{attribute 'GeneratedUsingTerminal: EL3024-0000-0019'}
{attribute addProperty BoxType "EL3024-0000-0019"}
{attribute addProperty Id "StatusAT %I*Status_F2CE6D917ValueAT %I*INT2"}
{attribute addProperty CRC "1245267073"}
{attribute addProperty Size "9"}
TYPE AI_Standard_Channel_4A394481 EXTENDS InputBase_8311D824 :
STRUCT
	{attribute addProperty Name "Status"}
	Status AT %I* : Status_F2CE6D91;
	{attribute addProperty Name "Value"}
	Value AT %I* : INT;
END_STRUCT
END_TYPE

(* stored: Version 1.2.0.0, ProductVersion 3.1.4024.9
   DUT AI_Standard_Channel_4A394481: Id {251797d0-b1b4-4c18-b943-2f317e61e5b1} *)
